// TIA Portal V20 export
DATA_BLOCK "ET500SP_513"   // DB278
// stored: MemoryReserve 100
   VAR
      "SP513.00 LEFT UNWINDER RADIUS SENSOR" : Int;
      "SP513.01 RIGHT UNWINDER RADIUS SENSOR" : Int;
      SPARE1 : Int;
      SPARE2 : Int;
   END_VAR
BEGIN
END_DATA_BLOCK
